// TIA Portal V17 export
// export: Created 2025-03-07T09:18:19.6203808Z, ExportSetting WithDefaults, DisplayName Totally Integrated Automation Portal, DisplayVersion V17 Update 8, DisplayName TIA Portal Openness, DisplayVersion V17 Update 8, DisplayName TIA Portal Version Control Interface, DisplayVersion V17, DisplayName SINAMICS Startdrive Advanced, DisplayVersion V17 SP2, DisplayName SINAMICS Startdrive G110M, G120, G120C, G120D, G120P, G115D, DisplayVersion V17 SP2, DisplayName SINAMICS Startdrive G130, G150, S120, S150, SINAMICS MV, S210, DisplayVersion V17 SP2, DisplayName STEP 7 Professional, DisplayVersion V17 Update 8, DisplayName SINUMERIK ONE STEP 7 Toolbox, DisplayVersion V17 Update 12, DisplayName SINUMERIK 840D sl STEP 7 Toolbox, DisplayVersion V17 Update 12, DisplayName STEP 7 Safety, DisplayVersion V17 Update 6, DisplayName WinCC Advanced, DisplayVersion V17 Update 8
FUNCTION "FC1701_KELLER_ASPIRATION_CONTROL" : Void   // FC1701, LAD
{ S7_Optimized_Access := 'TRUE' }
VERSION : 0.1
// stored: AutoNumber false, IsIECCheckEnabled false, SetENOAutomatically false, UDAEnableTagReadback false
   VAR CONSTANT
      FC_NUMBER : DInt := 1701;
   END_VAR
   VAR_TEMP   // added for the SCL form of the ladder/FBD networks
      _w1 : Bool;
      _s5time1 : S5Time;
   END_VAR
BEGIN

REGION Network 1: <<<<<<<<<<<<<<<<<<<< ASPIRATION CONTROL >>>>>>>>>>>>>>>>>>>>
END_REGION

REGION Network 2: KELLER ASPIRATION CONTROL CALL FB1701_KELLER_ASPIRATION_CONTROL
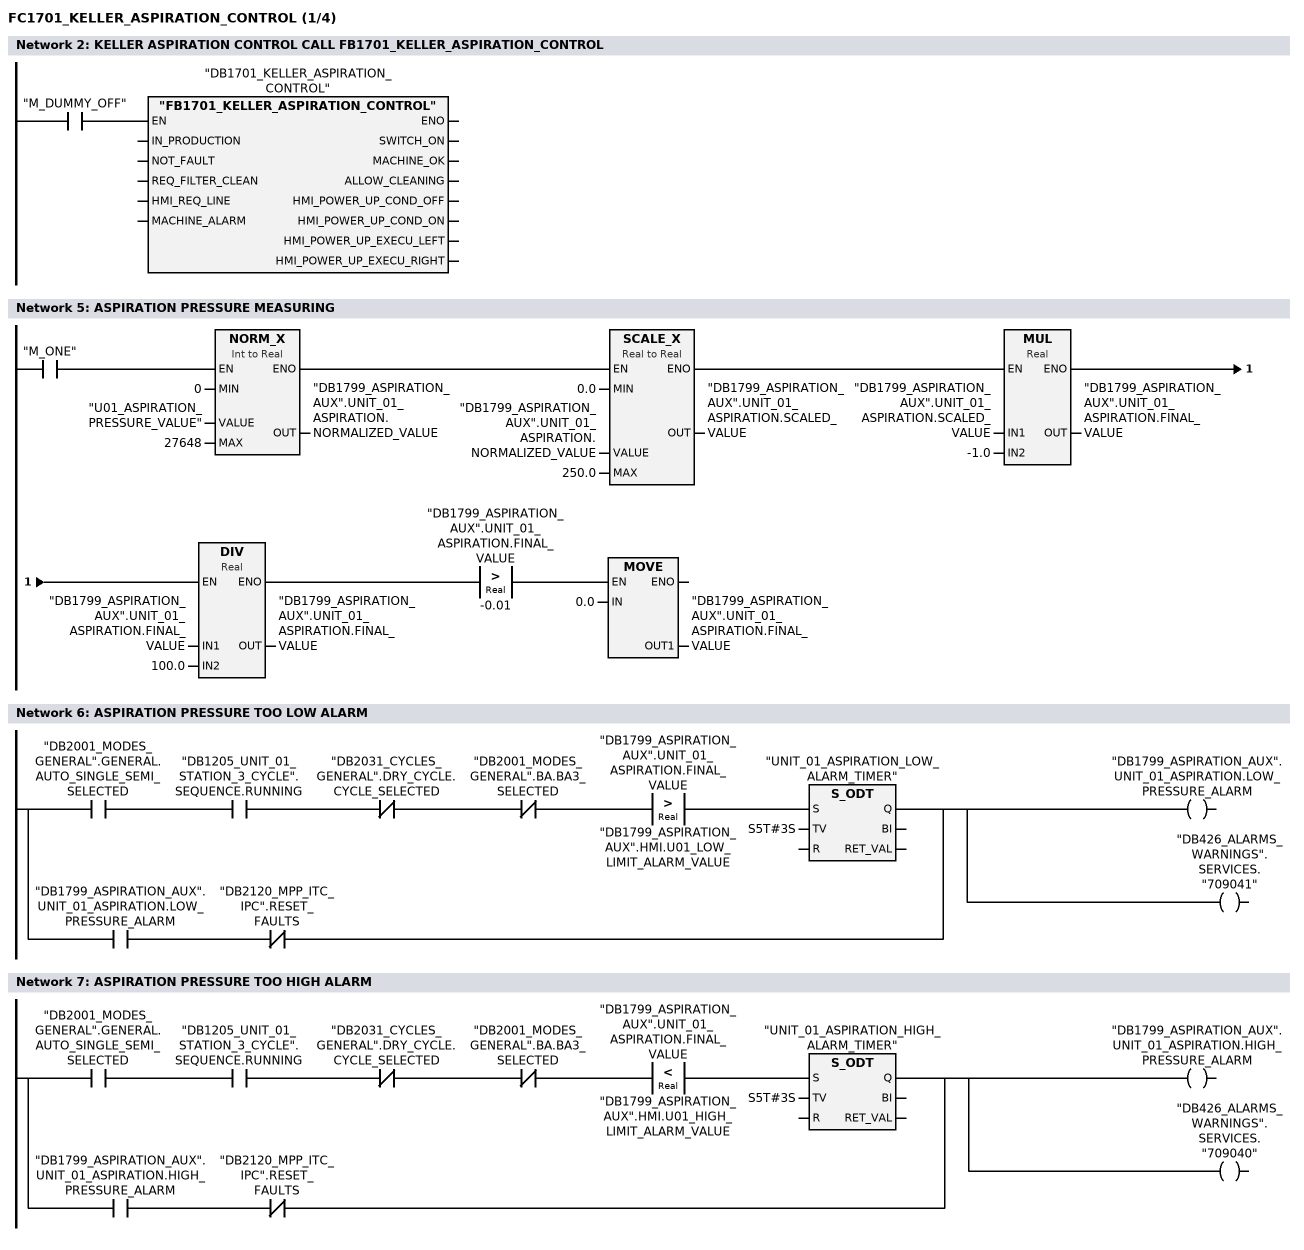
   RUNG wire#powerrail
      Contact( "M_DUMMY_OFF" )
      "DB1701_KELLER_ASPIRATION_CONTROL"(IN_PRODUCTION :=, NOT_FAULT :=, REQ_FILTER_CLEAN :=, HMI_REQ_LINE :=, MACHINE_ALARM :=, SWITCH_ON =>, MACHINE_OK =>, ALLOW_CLEANING =>, HMI_POWER_UP_COND_OFF =>, HMI_POWER_UP_COND_ON =>, HMI_POWER_UP_EXECU_LEFT =>, HMI_POWER_UP_EXECU_RIGHT =>)
   END_RUNG
   // the same network as SCL:
   IF "M_DUMMY_OFF" THEN
       "DB1701_KELLER_ASPIRATION_CONTROL"();   // "FB1701_KELLER_ASPIRATION_CONTROL"
   END_IF;
END_REGION

REGION Network 3: <<<<<<<<<<<<<<<<<<<< ASPIRTION CONTROL ALARMS >>>>>>>>>>>>>>>>>>>>
END_REGION

REGION Network 4: <<<<<<<<<<<<<<<<<<<<<<<<<<< UNIT 01 >>>>>>>>>>>>>>>>>>>>>>>>>>>
END_REGION

REGION Network 5: ASPIRATION PRESSURE MEASURING
   RUNG wire#powerrail
      Contact( "M_ONE" )
      { S7_Templates := "[SrcType := Int, DestType := Real]" } Normalize(min := 0, value := "U01_ASPIRATION_PRESSURE_VALUE", max := 27648, out => "DB1799_ASPIRATION_AUX".UNIT_01_ASPIRATION.NORMALIZED_VALUE)
      { S7_Templates := "[SrcType := Real, DestType := Real]" } Scale(min := 0.0, value := "DB1799_ASPIRATION_AUX".UNIT_01_ASPIRATION.NORMALIZED_VALUE, max := 250.0, out => "DB1799_ASPIRATION_AUX".UNIT_01_ASPIRATION.SCALED_VALUE)
      { S7_Templates := "SrcType := Real" } Mul(in1 := "DB1799_ASPIRATION_AUX".UNIT_01_ASPIRATION.SCALED_VALUE, in2 := -1.0, out => "DB1799_ASPIRATION_AUX".UNIT_01_ASPIRATION.FINAL_VALUE)
      { S7_Templates := "SrcType := Real" } Div(in1 := "DB1799_ASPIRATION_AUX".UNIT_01_ASPIRATION.FINAL_VALUE, in2 := 100.0, out => "DB1799_ASPIRATION_AUX".UNIT_01_ASPIRATION.FINAL_VALUE)
      { S7_Templates := "SrcType := Real" } GT_Contact(in1 := "DB1799_ASPIRATION_AUX".UNIT_01_ASPIRATION.FINAL_VALUE, in2 := -0.01)
      Move(in := 0.0, out1 => "DB1799_ASPIRATION_AUX".UNIT_01_ASPIRATION.FINAL_VALUE)
   END_RUNG
   // the same network as SCL:
   IF "M_ONE" THEN
       "DB1799_ASPIRATION_AUX".UNIT_01_ASPIRATION.NORMALIZED_VALUE := NORM_X(MIN := 0, VALUE := "U01_ASPIRATION_PRESSURE_VALUE", MAX := 27648);
       "DB1799_ASPIRATION_AUX".UNIT_01_ASPIRATION.SCALED_VALUE := SCALE_X(MIN := 0.0, VALUE := "DB1799_ASPIRATION_AUX".UNIT_01_ASPIRATION.NORMALIZED_VALUE, MAX := 250.0);
       "DB1799_ASPIRATION_AUX".UNIT_01_ASPIRATION.FINAL_VALUE := "DB1799_ASPIRATION_AUX".UNIT_01_ASPIRATION.SCALED_VALUE * (-1.0);
       "DB1799_ASPIRATION_AUX".UNIT_01_ASPIRATION.FINAL_VALUE := "DB1799_ASPIRATION_AUX".UNIT_01_ASPIRATION.FINAL_VALUE / 100.0;
   END_IF;
   IF "M_ONE" AND ("DB1799_ASPIRATION_AUX".UNIT_01_ASPIRATION.FINAL_VALUE > (-0.01)) THEN
       "DB1799_ASPIRATION_AUX".UNIT_01_ASPIRATION.FINAL_VALUE := 0.0;
   END_IF;
END_REGION

REGION Network 6: ASPIRATION PRESSURE TOO LOW ALARM
   RUNG wire#powerrail
      Contact( "DB2001_MODES_GENERAL".GENERAL.AUTO_SINGLE_SEMI_SELECTED )
      Contact( "DB1205_UNIT_01_STATION_3_CYCLE".SEQUENCE.RUNNING )
      I_Contact( "DB2031_CYCLES_GENERAL".DRY_CYCLE.CYCLE_SELECTED )
      I_Contact( "DB2001_MODES_GENERAL".BA.BA3_SELECTED )
      { S7_Templates := "SrcType := Real" } GT_Contact(in1 := "DB1799_ASPIRATION_AUX".UNIT_01_ASPIRATION.FINAL_VALUE, in2 := "DB1799_ASPIRATION_AUX".HMI.U01_LOW_LIMIT_ALARM_VALUE)
      S_ODT(T_NO := "UNIT_01_ASPIRATION_LOW_ALARM_TIMER", TV := S5T#3S, R :=, BI =>, RET_VAL =>)
      wire#w1
      Coil( "DB1799_ASPIRATION_AUX".UNIT_01_ASPIRATION.LOW_PRESSURE_ALARM )
   END_RUNG
   RUNG wire#powerrail
      Contact( "DB1799_ASPIRATION_AUX".UNIT_01_ASPIRATION.LOW_PRESSURE_ALARM )
      I_Contact( "DB2120_MPP_ITC_IPC".RESET_FAULTS )
   END_RUNG wire#w1
   RUNG wire#w1
      Coil( "DB426_ALARMS_WARNINGS".SERVICES."709041" )
   END_RUNG
   // the same network as SCL:
   #_s5time1 := S_ODT(T_NO := "UNIT_01_ASPIRATION_LOW_ALARM_TIMER",
                      S := "DB2001_MODES_GENERAL".GENERAL.AUTO_SINGLE_SEMI_SELECTED AND "DB1205_UNIT_01_STATION_3_CYCLE".SEQUENCE.RUNNING AND NOT "DB2031_CYCLES_GENERAL".DRY_CYCLE.CYCLE_SELECTED AND NOT "DB2001_MODES_GENERAL".BA.BA3_SELECTED AND ("DB1799_ASPIRATION_AUX".UNIT_01_ASPIRATION.FINAL_VALUE > "DB1799_ASPIRATION_AUX".HMI.U01_LOW_LIMIT_ALARM_VALUE),
                      TV := S5T#3S,
                      Q => #_w1);
   "DB1799_ASPIRATION_AUX".UNIT_01_ASPIRATION.LOW_PRESSURE_ALARM := #_w1 OR ("DB1799_ASPIRATION_AUX".UNIT_01_ASPIRATION.LOW_PRESSURE_ALARM AND NOT "DB2120_MPP_ITC_IPC".RESET_FAULTS);
   "DB426_ALARMS_WARNINGS".SERVICES."709041" := "DB1799_ASPIRATION_AUX".UNIT_01_ASPIRATION.LOW_PRESSURE_ALARM;
END_REGION

REGION Network 7: ASPIRATION PRESSURE TOO HIGH ALARM
   RUNG wire#powerrail
      Contact( "DB2001_MODES_GENERAL".GENERAL.AUTO_SINGLE_SEMI_SELECTED )
      Contact( "DB1205_UNIT_01_STATION_3_CYCLE".SEQUENCE.RUNNING )
      I_Contact( "DB2031_CYCLES_GENERAL".DRY_CYCLE.CYCLE_SELECTED )
      I_Contact( "DB2001_MODES_GENERAL".BA.BA3_SELECTED )
      { S7_Templates := "SrcType := Real" } LT_Contact(in1 := "DB1799_ASPIRATION_AUX".UNIT_01_ASPIRATION.FINAL_VALUE, in2 := "DB1799_ASPIRATION_AUX".HMI.U01_HIGH_LIMIT_ALARM_VALUE)
      S_ODT(T_NO := "UNIT_01_ASPIRATION_HIGH_ALARM_TIMER", TV := S5T#3S, R :=, BI =>, RET_VAL =>)
      wire#w1
      Coil( "DB1799_ASPIRATION_AUX".UNIT_01_ASPIRATION.HIGH_PRESSURE_ALARM )
   END_RUNG
   RUNG wire#powerrail
      Contact( "DB1799_ASPIRATION_AUX".UNIT_01_ASPIRATION.HIGH_PRESSURE_ALARM )
      I_Contact( "DB2120_MPP_ITC_IPC".RESET_FAULTS )
   END_RUNG wire#w1
   RUNG wire#w1
      Coil( "DB426_ALARMS_WARNINGS".SERVICES."709040" )
   END_RUNG
   // the same network as SCL:
   #_s5time1 := S_ODT(T_NO := "UNIT_01_ASPIRATION_HIGH_ALARM_TIMER",
                      S := "DB2001_MODES_GENERAL".GENERAL.AUTO_SINGLE_SEMI_SELECTED AND "DB1205_UNIT_01_STATION_3_CYCLE".SEQUENCE.RUNNING AND NOT "DB2031_CYCLES_GENERAL".DRY_CYCLE.CYCLE_SELECTED AND NOT "DB2001_MODES_GENERAL".BA.BA3_SELECTED AND ("DB1799_ASPIRATION_AUX".UNIT_01_ASPIRATION.FINAL_VALUE < "DB1799_ASPIRATION_AUX".HMI.U01_HIGH_LIMIT_ALARM_VALUE),
                      TV := S5T#3S,
                      Q => #_w1);
   "DB1799_ASPIRATION_AUX".UNIT_01_ASPIRATION.HIGH_PRESSURE_ALARM := #_w1 OR ("DB1799_ASPIRATION_AUX".UNIT_01_ASPIRATION.HIGH_PRESSURE_ALARM AND NOT "DB2120_MPP_ITC_IPC".RESET_FAULTS);
   "DB426_ALARMS_WARNINGS".SERVICES."709040" := "DB1799_ASPIRATION_AUX".UNIT_01_ASPIRATION.HIGH_PRESSURE_ALARM;
END_REGION

REGION Network 8: ASPIRATION PRESSURE TOO LOW WARNING
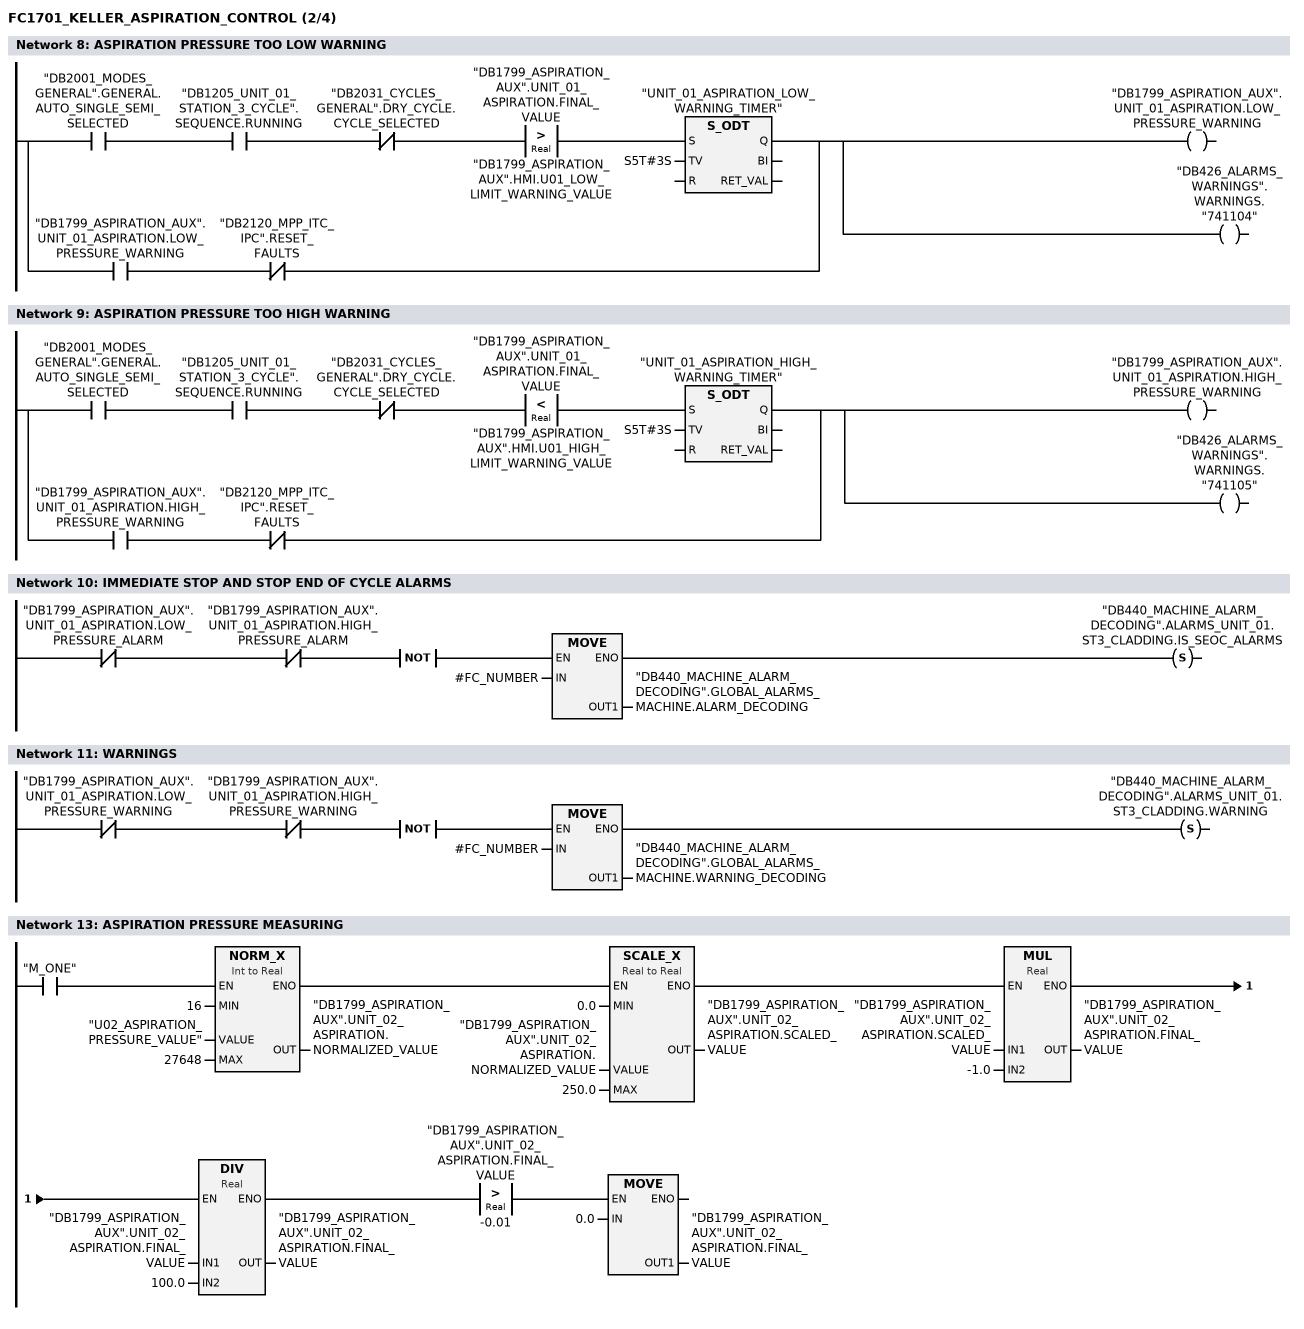
   RUNG wire#powerrail
      Contact( "DB2001_MODES_GENERAL".GENERAL.AUTO_SINGLE_SEMI_SELECTED )
      Contact( "DB1205_UNIT_01_STATION_3_CYCLE".SEQUENCE.RUNNING )
      I_Contact( "DB2031_CYCLES_GENERAL".DRY_CYCLE.CYCLE_SELECTED )
      { S7_Templates := "SrcType := Real" } GT_Contact(in1 := "DB1799_ASPIRATION_AUX".UNIT_01_ASPIRATION.FINAL_VALUE, in2 := "DB1799_ASPIRATION_AUX".HMI.U01_LOW_LIMIT_WARNING_VALUE)
      S_ODT(T_NO := "UNIT_01_ASPIRATION_LOW_WARNING_TIMER", TV := S5T#3S, R :=, BI =>, RET_VAL =>)
      wire#w1
      Coil( "DB1799_ASPIRATION_AUX".UNIT_01_ASPIRATION.LOW_PRESSURE_WARNING )
   END_RUNG
   RUNG wire#powerrail
      Contact( "DB1799_ASPIRATION_AUX".UNIT_01_ASPIRATION.LOW_PRESSURE_WARNING )
      I_Contact( "DB2120_MPP_ITC_IPC".RESET_FAULTS )
   END_RUNG wire#w1
   RUNG wire#w1
      Coil( "DB426_ALARMS_WARNINGS".WARNINGS."741104" )
   END_RUNG
   // the same network as SCL:
   #_s5time1 := S_ODT(T_NO := "UNIT_01_ASPIRATION_LOW_WARNING_TIMER",
                      S := "DB2001_MODES_GENERAL".GENERAL.AUTO_SINGLE_SEMI_SELECTED AND "DB1205_UNIT_01_STATION_3_CYCLE".SEQUENCE.RUNNING AND NOT "DB2031_CYCLES_GENERAL".DRY_CYCLE.CYCLE_SELECTED AND ("DB1799_ASPIRATION_AUX".UNIT_01_ASPIRATION.FINAL_VALUE > "DB1799_ASPIRATION_AUX".HMI.U01_LOW_LIMIT_WARNING_VALUE),
                      TV := S5T#3S,
                      Q => #_w1);
   "DB1799_ASPIRATION_AUX".UNIT_01_ASPIRATION.LOW_PRESSURE_WARNING := #_w1 OR ("DB1799_ASPIRATION_AUX".UNIT_01_ASPIRATION.LOW_PRESSURE_WARNING AND NOT "DB2120_MPP_ITC_IPC".RESET_FAULTS);
   "DB426_ALARMS_WARNINGS".WARNINGS."741104" := "DB1799_ASPIRATION_AUX".UNIT_01_ASPIRATION.LOW_PRESSURE_WARNING;
END_REGION

REGION Network 9: ASPIRATION PRESSURE TOO HIGH WARNING
   RUNG wire#powerrail
      Contact( "DB2001_MODES_GENERAL".GENERAL.AUTO_SINGLE_SEMI_SELECTED )
      Contact( "DB1205_UNIT_01_STATION_3_CYCLE".SEQUENCE.RUNNING )
      I_Contact( "DB2031_CYCLES_GENERAL".DRY_CYCLE.CYCLE_SELECTED )
      { S7_Templates := "SrcType := Real" } LT_Contact(in1 := "DB1799_ASPIRATION_AUX".UNIT_01_ASPIRATION.FINAL_VALUE, in2 := "DB1799_ASPIRATION_AUX".HMI.U01_HIGH_LIMIT_WARNING_VALUE)
      S_ODT(T_NO := "UNIT_01_ASPIRATION_HIGH_WARNING_TIMER", TV := S5T#3S, R :=, BI =>, RET_VAL =>)
      wire#w1
      Coil( "DB1799_ASPIRATION_AUX".UNIT_01_ASPIRATION.HIGH_PRESSURE_WARNING )
   END_RUNG
   RUNG wire#powerrail
      Contact( "DB1799_ASPIRATION_AUX".UNIT_01_ASPIRATION.HIGH_PRESSURE_WARNING )
      I_Contact( "DB2120_MPP_ITC_IPC".RESET_FAULTS )
   END_RUNG wire#w1
   RUNG wire#w1
      Coil( "DB426_ALARMS_WARNINGS".WARNINGS."741105" )
   END_RUNG
   // the same network as SCL:
   #_s5time1 := S_ODT(T_NO := "UNIT_01_ASPIRATION_HIGH_WARNING_TIMER",
                      S := "DB2001_MODES_GENERAL".GENERAL.AUTO_SINGLE_SEMI_SELECTED AND "DB1205_UNIT_01_STATION_3_CYCLE".SEQUENCE.RUNNING AND NOT "DB2031_CYCLES_GENERAL".DRY_CYCLE.CYCLE_SELECTED AND ("DB1799_ASPIRATION_AUX".UNIT_01_ASPIRATION.FINAL_VALUE < "DB1799_ASPIRATION_AUX".HMI.U01_HIGH_LIMIT_WARNING_VALUE),
                      TV := S5T#3S,
                      Q => #_w1);
   "DB1799_ASPIRATION_AUX".UNIT_01_ASPIRATION.HIGH_PRESSURE_WARNING := #_w1 OR ("DB1799_ASPIRATION_AUX".UNIT_01_ASPIRATION.HIGH_PRESSURE_WARNING AND NOT "DB2120_MPP_ITC_IPC".RESET_FAULTS);
   "DB426_ALARMS_WARNINGS".WARNINGS."741105" := "DB1799_ASPIRATION_AUX".UNIT_01_ASPIRATION.HIGH_PRESSURE_WARNING;
END_REGION

REGION Network 10: IMMEDIATE STOP AND STOP END OF CYCLE ALARMS
   RUNG wire#powerrail
      I_Contact( "DB1799_ASPIRATION_AUX".UNIT_01_ASPIRATION.LOW_PRESSURE_ALARM )
      I_Contact( "DB1799_ASPIRATION_AUX".UNIT_01_ASPIRATION.HIGH_PRESSURE_ALARM )
      Not()
      { S7_GenerateENO := "TRUE" } Move(in := #FC_NUMBER, out1 => "DB440_MACHINE_ALARM_DECODING".GLOBAL_ALARMS_MACHINE.ALARM_DECODING)
      S_Coil( "DB440_MACHINE_ALARM_DECODING".ALARMS_UNIT_01.ST3_CLADDING.IS_SEOC_ALARMS )
   END_RUNG
   // the same network as SCL:
   // ENO of a box is taken as its EN; it also drops when the box reports an error
   IF NOT (NOT "DB1799_ASPIRATION_AUX".UNIT_01_ASPIRATION.LOW_PRESSURE_ALARM AND NOT "DB1799_ASPIRATION_AUX".UNIT_01_ASPIRATION.HIGH_PRESSURE_ALARM) THEN
       "DB440_MACHINE_ALARM_DECODING".GLOBAL_ALARMS_MACHINE.ALARM_DECODING := #FC_NUMBER;
       "DB440_MACHINE_ALARM_DECODING".ALARMS_UNIT_01.ST3_CLADDING.IS_SEOC_ALARMS := TRUE;
   END_IF;
END_REGION

REGION Network 11: WARNINGS
   RUNG wire#powerrail
      I_Contact( "DB1799_ASPIRATION_AUX".UNIT_01_ASPIRATION.LOW_PRESSURE_WARNING )
      I_Contact( "DB1799_ASPIRATION_AUX".UNIT_01_ASPIRATION.HIGH_PRESSURE_WARNING )
      Not()
      Move(in := #FC_NUMBER, out1 => "DB440_MACHINE_ALARM_DECODING".GLOBAL_ALARMS_MACHINE.WARNING_DECODING)
      S_Coil( "DB440_MACHINE_ALARM_DECODING".ALARMS_UNIT_01.ST3_CLADDING.WARNING )
   END_RUNG
   // the same network as SCL:
   IF NOT (NOT "DB1799_ASPIRATION_AUX".UNIT_01_ASPIRATION.LOW_PRESSURE_WARNING AND NOT "DB1799_ASPIRATION_AUX".UNIT_01_ASPIRATION.HIGH_PRESSURE_WARNING) THEN
       "DB440_MACHINE_ALARM_DECODING".GLOBAL_ALARMS_MACHINE.WARNING_DECODING := #FC_NUMBER;
       "DB440_MACHINE_ALARM_DECODING".ALARMS_UNIT_01.ST3_CLADDING.WARNING := TRUE;
   END_IF;
END_REGION

REGION Network 12: <<<<<<<<<<<<<<<<<<<<<<<<<<< UNIT 02 >>>>>>>>>>>>>>>>>>>>>>>>>>>
END_REGION

REGION Network 13: ASPIRATION PRESSURE MEASURING
   RUNG wire#powerrail
      Contact( "M_ONE" )
      { S7_Templates := "[SrcType := Int, DestType := Real]" } Normalize(min := 16, value := "U02_ASPIRATION_PRESSURE_VALUE", max := 27648, out => "DB1799_ASPIRATION_AUX".UNIT_02_ASPIRATION.NORMALIZED_VALUE)
      { S7_Templates := "[SrcType := Real, DestType := Real]" } Scale(min := 0.0, value := "DB1799_ASPIRATION_AUX".UNIT_02_ASPIRATION.NORMALIZED_VALUE, max := 250.0, out => "DB1799_ASPIRATION_AUX".UNIT_02_ASPIRATION.SCALED_VALUE)
      { S7_Templates := "SrcType := Real" } Mul(in1 := "DB1799_ASPIRATION_AUX".UNIT_02_ASPIRATION.SCALED_VALUE, in2 := -1.0, out => "DB1799_ASPIRATION_AUX".UNIT_02_ASPIRATION.FINAL_VALUE)
      { S7_Templates := "SrcType := Real" } Div(in1 := "DB1799_ASPIRATION_AUX".UNIT_02_ASPIRATION.FINAL_VALUE, in2 := 100.0, out => "DB1799_ASPIRATION_AUX".UNIT_02_ASPIRATION.FINAL_VALUE)
      { S7_Templates := "SrcType := Real" } GT_Contact(in1 := "DB1799_ASPIRATION_AUX".UNIT_02_ASPIRATION.FINAL_VALUE, in2 := -0.01)
      Move(in := 0.0, out1 => "DB1799_ASPIRATION_AUX".UNIT_02_ASPIRATION.FINAL_VALUE)
   END_RUNG
   // the same network as SCL:
   IF "M_ONE" THEN
       "DB1799_ASPIRATION_AUX".UNIT_02_ASPIRATION.NORMALIZED_VALUE := NORM_X(MIN := 16, VALUE := "U02_ASPIRATION_PRESSURE_VALUE", MAX := 27648);
       "DB1799_ASPIRATION_AUX".UNIT_02_ASPIRATION.SCALED_VALUE := SCALE_X(MIN := 0.0, VALUE := "DB1799_ASPIRATION_AUX".UNIT_02_ASPIRATION.NORMALIZED_VALUE, MAX := 250.0);
       "DB1799_ASPIRATION_AUX".UNIT_02_ASPIRATION.FINAL_VALUE := "DB1799_ASPIRATION_AUX".UNIT_02_ASPIRATION.SCALED_VALUE * (-1.0);
       "DB1799_ASPIRATION_AUX".UNIT_02_ASPIRATION.FINAL_VALUE := "DB1799_ASPIRATION_AUX".UNIT_02_ASPIRATION.FINAL_VALUE / 100.0;
   END_IF;
   IF "M_ONE" AND ("DB1799_ASPIRATION_AUX".UNIT_02_ASPIRATION.FINAL_VALUE > (-0.01)) THEN
       "DB1799_ASPIRATION_AUX".UNIT_02_ASPIRATION.FINAL_VALUE := 0.0;
   END_IF;
END_REGION

REGION Network 14: ASPIRATION PRESSURE TOO LOW ALARM
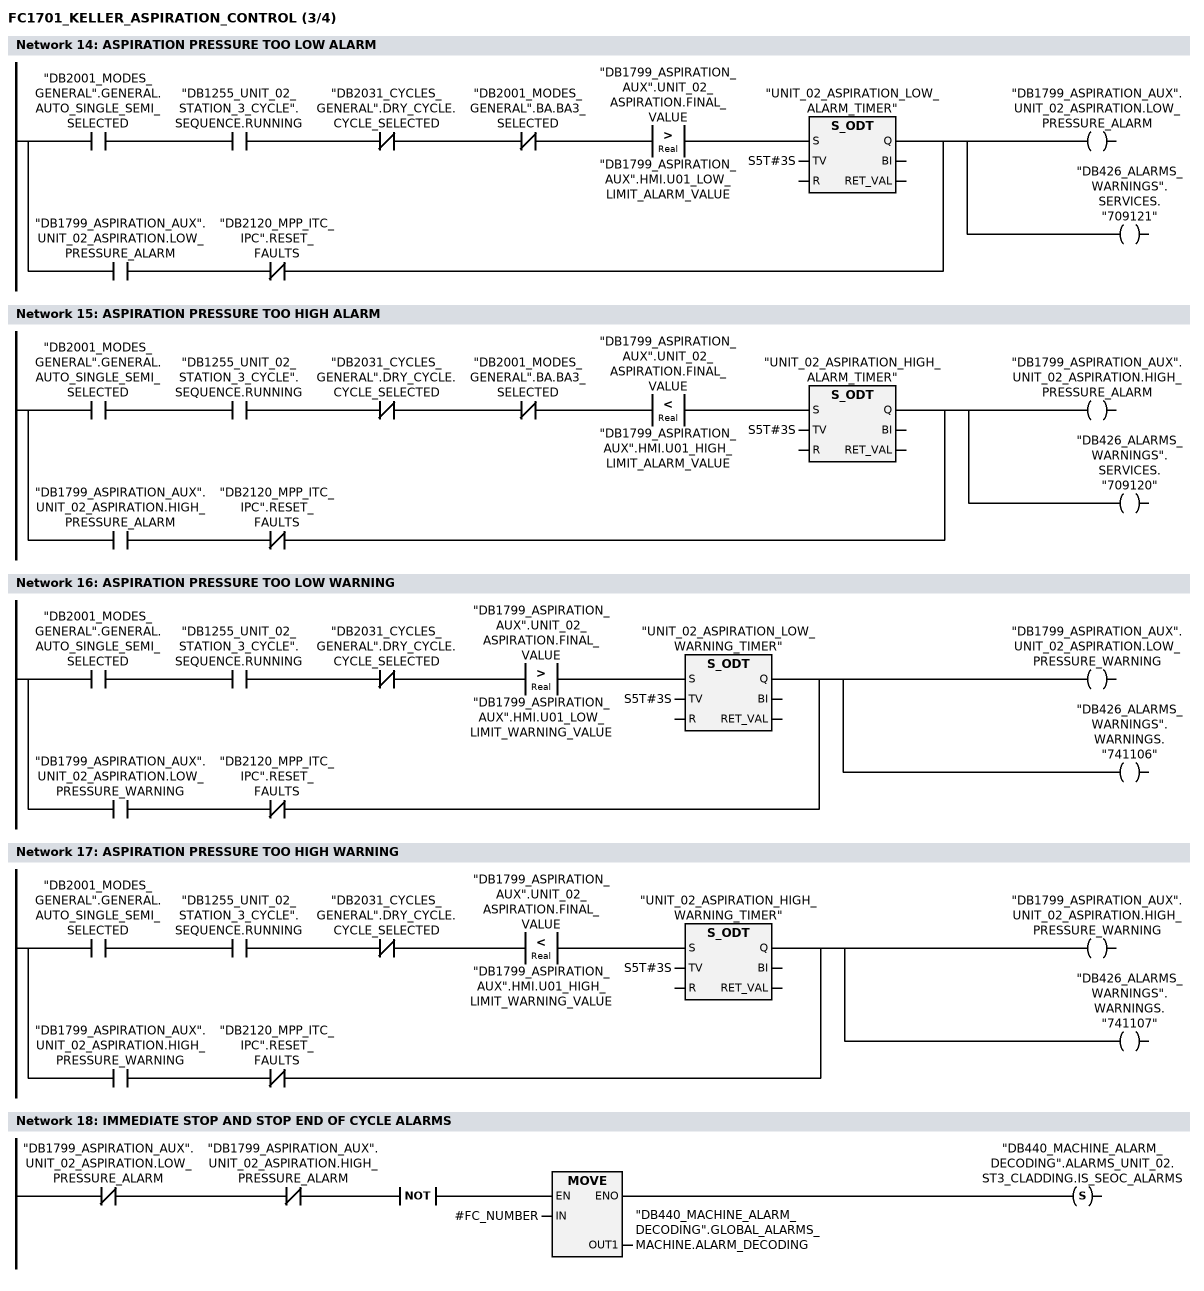
   RUNG wire#powerrail
      Contact( "DB2001_MODES_GENERAL".GENERAL.AUTO_SINGLE_SEMI_SELECTED )
      Contact( "DB1255_UNIT_02_STATION_3_CYCLE".SEQUENCE.RUNNING )
      I_Contact( "DB2031_CYCLES_GENERAL".DRY_CYCLE.CYCLE_SELECTED )
      I_Contact( "DB2001_MODES_GENERAL".BA.BA3_SELECTED )
      { S7_Templates := "SrcType := Real" } GT_Contact(in1 := "DB1799_ASPIRATION_AUX".UNIT_02_ASPIRATION.FINAL_VALUE, in2 := "DB1799_ASPIRATION_AUX".HMI.U01_LOW_LIMIT_ALARM_VALUE)
      S_ODT(T_NO := "UNIT_02_ASPIRATION_LOW_ALARM_TIMER", TV := S5T#3S, R :=, BI =>, RET_VAL =>)
      wire#w1
      Coil( "DB1799_ASPIRATION_AUX".UNIT_02_ASPIRATION.LOW_PRESSURE_ALARM )
   END_RUNG
   RUNG wire#powerrail
      Contact( "DB1799_ASPIRATION_AUX".UNIT_02_ASPIRATION.LOW_PRESSURE_ALARM )
      I_Contact( "DB2120_MPP_ITC_IPC".RESET_FAULTS )
   END_RUNG wire#w1
   RUNG wire#w1
      Coil( "DB426_ALARMS_WARNINGS".SERVICES."709121" )
   END_RUNG
   // the same network as SCL:
   #_s5time1 := S_ODT(T_NO := "UNIT_02_ASPIRATION_LOW_ALARM_TIMER",
                      S := "DB2001_MODES_GENERAL".GENERAL.AUTO_SINGLE_SEMI_SELECTED AND "DB1255_UNIT_02_STATION_3_CYCLE".SEQUENCE.RUNNING AND NOT "DB2031_CYCLES_GENERAL".DRY_CYCLE.CYCLE_SELECTED AND NOT "DB2001_MODES_GENERAL".BA.BA3_SELECTED AND ("DB1799_ASPIRATION_AUX".UNIT_02_ASPIRATION.FINAL_VALUE > "DB1799_ASPIRATION_AUX".HMI.U01_LOW_LIMIT_ALARM_VALUE),
                      TV := S5T#3S,
                      Q => #_w1);
   "DB1799_ASPIRATION_AUX".UNIT_02_ASPIRATION.LOW_PRESSURE_ALARM := #_w1 OR ("DB1799_ASPIRATION_AUX".UNIT_02_ASPIRATION.LOW_PRESSURE_ALARM AND NOT "DB2120_MPP_ITC_IPC".RESET_FAULTS);
   "DB426_ALARMS_WARNINGS".SERVICES."709121" := "DB1799_ASPIRATION_AUX".UNIT_02_ASPIRATION.LOW_PRESSURE_ALARM;
END_REGION

REGION Network 15: ASPIRATION PRESSURE TOO HIGH ALARM
   RUNG wire#powerrail
      Contact( "DB2001_MODES_GENERAL".GENERAL.AUTO_SINGLE_SEMI_SELECTED )
      Contact( "DB1255_UNIT_02_STATION_3_CYCLE".SEQUENCE.RUNNING )
      I_Contact( "DB2031_CYCLES_GENERAL".DRY_CYCLE.CYCLE_SELECTED )
      I_Contact( "DB2001_MODES_GENERAL".BA.BA3_SELECTED )
      { S7_Templates := "SrcType := Real" } LT_Contact(in1 := "DB1799_ASPIRATION_AUX".UNIT_02_ASPIRATION.FINAL_VALUE, in2 := "DB1799_ASPIRATION_AUX".HMI.U01_HIGH_LIMIT_ALARM_VALUE)
      S_ODT(T_NO := "UNIT_02_ASPIRATION_HIGH_ALARM_TIMER", TV := S5T#3S, R :=, BI =>, RET_VAL =>)
      wire#w1
      Coil( "DB1799_ASPIRATION_AUX".UNIT_02_ASPIRATION.HIGH_PRESSURE_ALARM )
   END_RUNG
   RUNG wire#powerrail
      Contact( "DB1799_ASPIRATION_AUX".UNIT_02_ASPIRATION.HIGH_PRESSURE_ALARM )
      I_Contact( "DB2120_MPP_ITC_IPC".RESET_FAULTS )
   END_RUNG wire#w1
   RUNG wire#w1
      Coil( "DB426_ALARMS_WARNINGS".SERVICES."709120" )
   END_RUNG
   // the same network as SCL:
   #_s5time1 := S_ODT(T_NO := "UNIT_02_ASPIRATION_HIGH_ALARM_TIMER",
                      S := "DB2001_MODES_GENERAL".GENERAL.AUTO_SINGLE_SEMI_SELECTED AND "DB1255_UNIT_02_STATION_3_CYCLE".SEQUENCE.RUNNING AND NOT "DB2031_CYCLES_GENERAL".DRY_CYCLE.CYCLE_SELECTED AND NOT "DB2001_MODES_GENERAL".BA.BA3_SELECTED AND ("DB1799_ASPIRATION_AUX".UNIT_02_ASPIRATION.FINAL_VALUE < "DB1799_ASPIRATION_AUX".HMI.U01_HIGH_LIMIT_ALARM_VALUE),
                      TV := S5T#3S,
                      Q => #_w1);
   "DB1799_ASPIRATION_AUX".UNIT_02_ASPIRATION.HIGH_PRESSURE_ALARM := #_w1 OR ("DB1799_ASPIRATION_AUX".UNIT_02_ASPIRATION.HIGH_PRESSURE_ALARM AND NOT "DB2120_MPP_ITC_IPC".RESET_FAULTS);
   "DB426_ALARMS_WARNINGS".SERVICES."709120" := "DB1799_ASPIRATION_AUX".UNIT_02_ASPIRATION.HIGH_PRESSURE_ALARM;
END_REGION

REGION Network 16: ASPIRATION PRESSURE TOO LOW WARNING
   RUNG wire#powerrail
      Contact( "DB2001_MODES_GENERAL".GENERAL.AUTO_SINGLE_SEMI_SELECTED )
      Contact( "DB1255_UNIT_02_STATION_3_CYCLE".SEQUENCE.RUNNING )
      I_Contact( "DB2031_CYCLES_GENERAL".DRY_CYCLE.CYCLE_SELECTED )
      { S7_Templates := "SrcType := Real" } GT_Contact(in1 := "DB1799_ASPIRATION_AUX".UNIT_02_ASPIRATION.FINAL_VALUE, in2 := "DB1799_ASPIRATION_AUX".HMI.U01_LOW_LIMIT_WARNING_VALUE)
      S_ODT(T_NO := "UNIT_02_ASPIRATION_LOW_WARNING_TIMER", TV := S5T#3S, R :=, BI =>, RET_VAL =>)
      wire#w1
      Coil( "DB1799_ASPIRATION_AUX".UNIT_02_ASPIRATION.LOW_PRESSURE_WARNING )
   END_RUNG
   RUNG wire#powerrail
      Contact( "DB1799_ASPIRATION_AUX".UNIT_02_ASPIRATION.LOW_PRESSURE_WARNING )
      I_Contact( "DB2120_MPP_ITC_IPC".RESET_FAULTS )
   END_RUNG wire#w1
   RUNG wire#w1
      Coil( "DB426_ALARMS_WARNINGS".WARNINGS."741106" )
   END_RUNG
   // the same network as SCL:
   #_s5time1 := S_ODT(T_NO := "UNIT_02_ASPIRATION_LOW_WARNING_TIMER",
                      S := "DB2001_MODES_GENERAL".GENERAL.AUTO_SINGLE_SEMI_SELECTED AND "DB1255_UNIT_02_STATION_3_CYCLE".SEQUENCE.RUNNING AND NOT "DB2031_CYCLES_GENERAL".DRY_CYCLE.CYCLE_SELECTED AND ("DB1799_ASPIRATION_AUX".UNIT_02_ASPIRATION.FINAL_VALUE > "DB1799_ASPIRATION_AUX".HMI.U01_LOW_LIMIT_WARNING_VALUE),
                      TV := S5T#3S,
                      Q => #_w1);
   "DB1799_ASPIRATION_AUX".UNIT_02_ASPIRATION.LOW_PRESSURE_WARNING := #_w1 OR ("DB1799_ASPIRATION_AUX".UNIT_02_ASPIRATION.LOW_PRESSURE_WARNING AND NOT "DB2120_MPP_ITC_IPC".RESET_FAULTS);
   "DB426_ALARMS_WARNINGS".WARNINGS."741106" := "DB1799_ASPIRATION_AUX".UNIT_02_ASPIRATION.LOW_PRESSURE_WARNING;
END_REGION

REGION Network 17: ASPIRATION PRESSURE TOO HIGH WARNING
   RUNG wire#powerrail
      Contact( "DB2001_MODES_GENERAL".GENERAL.AUTO_SINGLE_SEMI_SELECTED )
      Contact( "DB1255_UNIT_02_STATION_3_CYCLE".SEQUENCE.RUNNING )
      I_Contact( "DB2031_CYCLES_GENERAL".DRY_CYCLE.CYCLE_SELECTED )
      { S7_Templates := "SrcType := Real" } LT_Contact(in1 := "DB1799_ASPIRATION_AUX".UNIT_02_ASPIRATION.FINAL_VALUE, in2 := "DB1799_ASPIRATION_AUX".HMI.U01_HIGH_LIMIT_WARNING_VALUE)
      S_ODT(T_NO := "UNIT_02_ASPIRATION_HIGH_WARNING_TIMER", TV := S5T#3S, R :=, BI =>, RET_VAL =>)
      wire#w1
      Coil( "DB1799_ASPIRATION_AUX".UNIT_02_ASPIRATION.HIGH_PRESSURE_WARNING )
   END_RUNG
   RUNG wire#powerrail
      Contact( "DB1799_ASPIRATION_AUX".UNIT_02_ASPIRATION.HIGH_PRESSURE_WARNING )
      I_Contact( "DB2120_MPP_ITC_IPC".RESET_FAULTS )
   END_RUNG wire#w1
   RUNG wire#w1
      Coil( "DB426_ALARMS_WARNINGS".WARNINGS."741107" )
   END_RUNG
   // the same network as SCL:
   #_s5time1 := S_ODT(T_NO := "UNIT_02_ASPIRATION_HIGH_WARNING_TIMER",
                      S := "DB2001_MODES_GENERAL".GENERAL.AUTO_SINGLE_SEMI_SELECTED AND "DB1255_UNIT_02_STATION_3_CYCLE".SEQUENCE.RUNNING AND NOT "DB2031_CYCLES_GENERAL".DRY_CYCLE.CYCLE_SELECTED AND ("DB1799_ASPIRATION_AUX".UNIT_02_ASPIRATION.FINAL_VALUE < "DB1799_ASPIRATION_AUX".HMI.U01_HIGH_LIMIT_WARNING_VALUE),
                      TV := S5T#3S,
                      Q => #_w1);
   "DB1799_ASPIRATION_AUX".UNIT_02_ASPIRATION.HIGH_PRESSURE_WARNING := #_w1 OR ("DB1799_ASPIRATION_AUX".UNIT_02_ASPIRATION.HIGH_PRESSURE_WARNING AND NOT "DB2120_MPP_ITC_IPC".RESET_FAULTS);
   "DB426_ALARMS_WARNINGS".WARNINGS."741107" := "DB1799_ASPIRATION_AUX".UNIT_02_ASPIRATION.HIGH_PRESSURE_WARNING;
END_REGION

REGION Network 18: IMMEDIATE STOP AND STOP END OF CYCLE ALARMS
   RUNG wire#powerrail
      I_Contact( "DB1799_ASPIRATION_AUX".UNIT_02_ASPIRATION.LOW_PRESSURE_ALARM )
      I_Contact( "DB1799_ASPIRATION_AUX".UNIT_02_ASPIRATION.HIGH_PRESSURE_ALARM )
      Not()
      { S7_GenerateENO := "TRUE" } Move(in := #FC_NUMBER, out1 => "DB440_MACHINE_ALARM_DECODING".GLOBAL_ALARMS_MACHINE.ALARM_DECODING)
      S_Coil( "DB440_MACHINE_ALARM_DECODING".ALARMS_UNIT_02.ST3_CLADDING.IS_SEOC_ALARMS )
   END_RUNG
   // the same network as SCL:
   // ENO of a box is taken as its EN; it also drops when the box reports an error
   IF NOT (NOT "DB1799_ASPIRATION_AUX".UNIT_02_ASPIRATION.LOW_PRESSURE_ALARM AND NOT "DB1799_ASPIRATION_AUX".UNIT_02_ASPIRATION.HIGH_PRESSURE_ALARM) THEN
       "DB440_MACHINE_ALARM_DECODING".GLOBAL_ALARMS_MACHINE.ALARM_DECODING := #FC_NUMBER;
       "DB440_MACHINE_ALARM_DECODING".ALARMS_UNIT_02.ST3_CLADDING.IS_SEOC_ALARMS := TRUE;
   END_IF;
END_REGION

REGION Network 19: WARNINGS
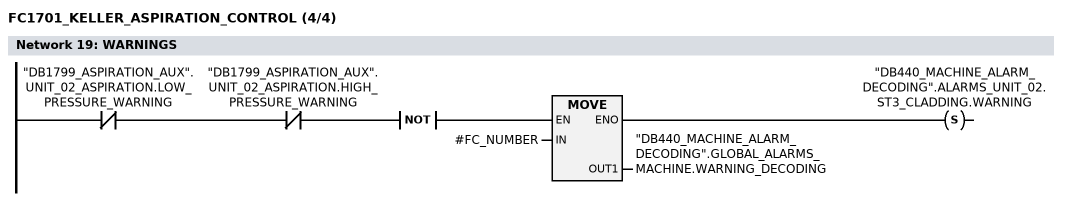
   RUNG wire#powerrail
      I_Contact( "DB1799_ASPIRATION_AUX".UNIT_02_ASPIRATION.LOW_PRESSURE_WARNING )
      I_Contact( "DB1799_ASPIRATION_AUX".UNIT_02_ASPIRATION.HIGH_PRESSURE_WARNING )
      Not()
      Move(in := #FC_NUMBER, out1 => "DB440_MACHINE_ALARM_DECODING".GLOBAL_ALARMS_MACHINE.WARNING_DECODING)
      S_Coil( "DB440_MACHINE_ALARM_DECODING".ALARMS_UNIT_02.ST3_CLADDING.WARNING )
   END_RUNG
   // the same network as SCL:
   IF NOT (NOT "DB1799_ASPIRATION_AUX".UNIT_02_ASPIRATION.LOW_PRESSURE_WARNING AND NOT "DB1799_ASPIRATION_AUX".UNIT_02_ASPIRATION.HIGH_PRESSURE_WARNING) THEN
       "DB440_MACHINE_ALARM_DECODING".GLOBAL_ALARMS_MACHINE.WARNING_DECODING := #FC_NUMBER;
       "DB440_MACHINE_ALARM_DECODING".ALARMS_UNIT_02.ST3_CLADDING.WARNING := TRUE;
   END_IF;
END_REGION
END_FUNCTION
